// Mitsubishi GX Works2 project: PLC-Servo 실습 과제 2   PLC: Q03UDV

PROGRAM MAIN
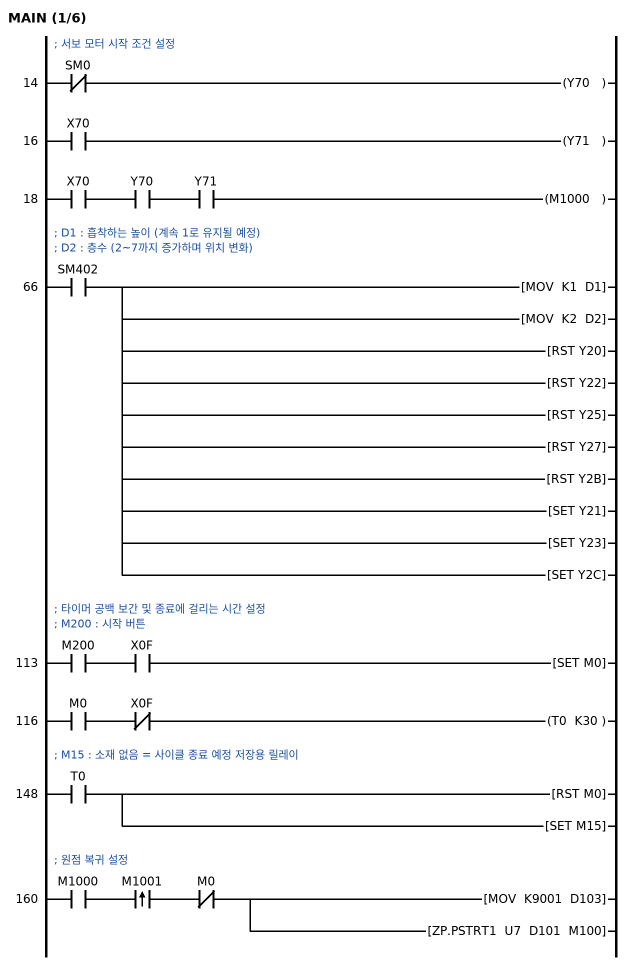
; 서보 모터 시작 조건 설정
14    LDI     SM0
      OUT     Y70
16    LD      X70
      OUT     Y71
18    LD      X70
      AND     Y70
      AND     Y71
      OUT     M1000
; D1 : 흡착하는 높이 (계속 1로 유지될 예정)
; D2 : 층수 (2~7까지 증가하며 위치 변화)
66    LD      SM402
      MOV     K1 D1
      MOV     K2 D2
      RST     Y20
      RST     Y22
      RST     Y25
      RST     Y27
      RST     Y2B
      SET     Y21
      SET     Y23
      SET     Y2C
; 타이머 공백 보간 및 종료에 걸리는 시간 설정
; M200 : 시작 버튼
113   LD      M200
      AND     X0F
      SET     M0
116   LD      M0
      ANI     X0F
      OUT     T0 K30
; M15 : 소재 없음 = 사이클 종료 예정 저장용 릴레이
148   LD      T0
      RST     M0
      SET     M15
; 원점 복귀 설정
160   LD      M1000
      ANDP    M1001
      ANI     M0
      MOV     K9001 D103
      ZP.PSTRT1 U7 D101 M100
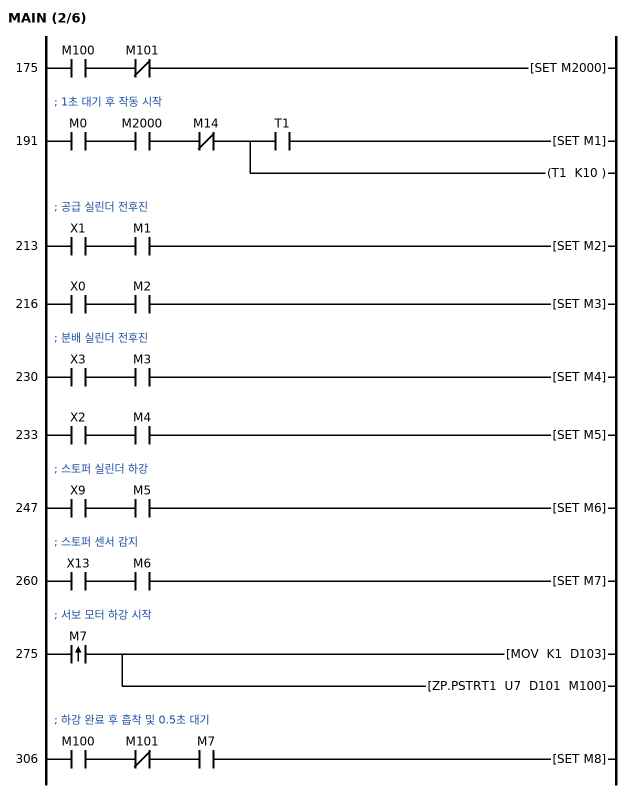
175   LD      M100
      ANI     M101
      SET     M2000
; 1초 대기 후 작동 시작
191   LD      M0
      AND     M2000
      ANI     M14
      MPS
      AND     T1
      SET     M1
      MPP
      OUT     T1 K10
; 공급 실린더 전후진
213   LD      X1
      AND     M1
      SET     M2
216   LD      X0
      AND     M2
      SET     M3
; 분배 실린더 전후진
230   LD      X3
      AND     M3
      SET     M4
233   LD      X2
      AND     M4
      SET     M5
; 스토퍼 실린더 하강
247   LD      X9
      AND     M5
      SET     M6
; 스토퍼 센서 감지
260   LD      X13
      AND     M6
      SET     M7
; 서보 모터 하강 시작
275   LDP     M7
      MOV     K1 D103
      ZP.PSTRT1 U7 D101 M100
; 하강 완료 후 흡착 및 0.5초 대기
306   LD      M100
      ANI     M101
      AND     M7
      SET     M8
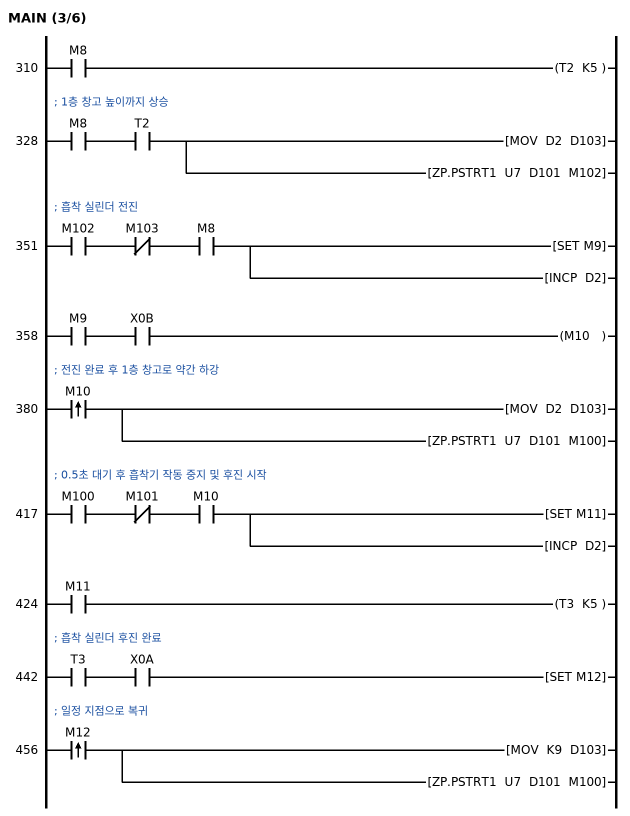
310   LD      M8
      OUT     T2 K5
; 1층 창고 높이까지 상승
328   LD      M8
      AND     T2
      MOV     D2 D103
      ZP.PSTRT1 U7 D101 M102
; 흡착 실린더 전진
351   LD      M102
      ANI     M103
      AND     M8
      SET     M9
      INCP    D2
358   LD      M9
      AND     X0B
      OUT     M10
; 전진 완료 후 1층 창고로 약간 하강
380   LDP     M10
      MOV     D2 D103
      ZP.PSTRT1 U7 D101 M100
; 0.5초 대기 후 흡착기 작동 중지 및 후진 시작
417   LD      M100
      ANI     M101
      AND     M10
      SET     M11
      INCP    D2
424   LD      M11
      OUT     T3 K5
; 흡착 실린더 후진 완료
442   LD      T3
      AND     X0A
      SET     M12
; 일정 지점으로 복귀
456   LDP     M12
      MOV     K9 D103
      ZP.PSTRT1 U7 D101 M100
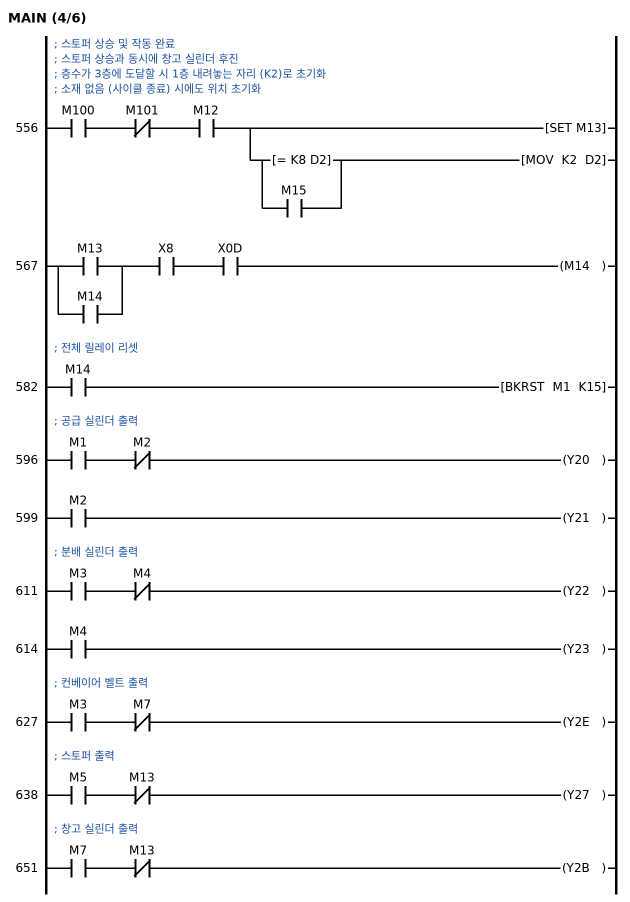
; 스토퍼 상승 및 작동 완료
; 스토퍼 상승과 동시에 창고 실린더 후진
; 층수가 3층에 도달할 시 1층 내려놓는 자리 (K2)로 초기화
; 소재 없음 (사이클 종료) 시에도 위치 초기화
556   LD      M100
      ANI     M101
      AND     M12
      SET     M13
      LD=     K8 D2
      OR      M15
      ANB
      MOV     K2 D2
567   LD      M13
      OR      M14
      AND     X8
      AND     X0D
      OUT     M14
; 전체 릴레이 리셋
582   LD      M14
      BKRST   M1 K15
; 공급 실린더 출력
596   LD      M1
      ANI     M2
      OUT     Y20
599   LD      M2
      OUT     Y21
; 분배 실린더 출력
611   LD      M3
      ANI     M4
      OUT     Y22
614   LD      M4
      OUT     Y23
; 컨베이어 벨트 출력
627   LD      M3
      ANI     M7
      OUT     Y2E
; 스토퍼 출력
638   LD      M5
      ANI     M13
      OUT     Y27
; 창고 실린더 출력
651   LD      M7
      ANI     M13
      OUT     Y2B
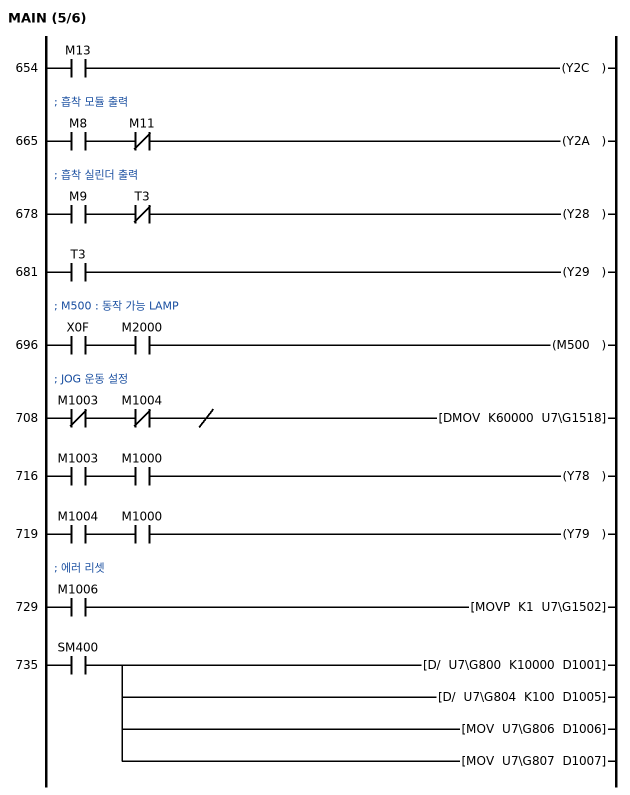
654   LD      M13
      OUT     Y2C
; 흡착 모듈 출력
665   LD      M8
      ANI     M11
      OUT     Y2A
; 흡착 실린더 출력
678   LD      M9
      ANI     T3
      OUT     Y28
681   LD      T3
      OUT     Y29
; M500 : 동작 가능 LAMP
696   LD      X0F
      AND     M2000
      OUT     M500
; JOG 운동 설정
708   LDI     M1003
      ANI     M1004
      INV
      DMOV    K60000 U7\G1518
716   LD      M1003
      AND     M1000
      OUT     Y78
719   LD      M1004
      AND     M1000
      OUT     Y79
; 에러 리셋
729   LD      M1006
      MOVP    K1 U7\G1502
735   LD      SM400
      D/      U7\G800 K10000 D1001
      D/      U7\G804 K100 D1005
      MOV     U7\G806 D1006
      MOV     U7\G807 D1007
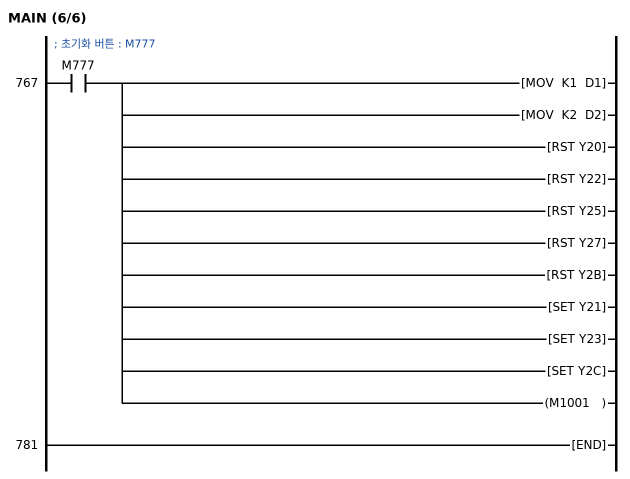
; 초기화 버튼 : M777
767   LD      M777
      MOV     K1 D1
      MOV     K2 D2
      RST     Y20
      RST     Y22
      RST     Y25
      RST     Y27
      RST     Y2B
      SET     Y21
      SET     Y23
      SET     Y2C
      OUT     M1001
781   END
END_PROGRAM
